{attribute addProperty BoxType "EK1960-2600-0021"}
{attribute addProperty Id "FSoE_CommandUSINT811FSOUT_Module_1_Module_FaultBIT10.1251FSOUT_Module_2_Module_FaultBIT10.1251FSOUT_Module_3_Module_FaultBIT10.1251FSOUT_Module_4_Module_FaultBIT10.1251FSOUT_Module_5_Module_FaultBIT10.1251FSOUT_Module_6_Module_FaultBIT10.1251FSOUT_Relais_Module_Module_FaultBIT10.1251FSIN_Module_1_Channel_1_Input_X6_1BIT10.1251FSIN_Module_1_Channel_2_Input_X6_2BIT10.1252FSIN_Module_1_Module_FaultBIT10.1251FSIN_Module_2_Channel_1_Input_X6_3BIT10.1251FSIN_Module_2_Channel_2_Input_X6_4BIT10.1252FSIN_Module_2_Module_FaultBIT10.1251FSIN_Module_3_Channel_1_Input_X6_5BIT10.1251FSIN_Module_3_Channel_2_Input_X6_6BIT10.1252FSIN_Module_3_Module_FaultBIT10.1251FSoE_CRC_000UINT1623FSIN_Module_4_Channel_1_Input_X6_7BIT10.1251FSIN_Module_4_Channel_2_Input_X6_8BIT10.1252FSIN_Module_4_Module_FaultBIT10.1251FSIN_Module_5_Channel_1_Input_X6_9BIT10.1251FSIN_Module_5_Channel_2_Input_X6_10BIT10.1252FSIN_Module_5_Module_FaultBIT10.1251FSIN_Module_6_Channel_1_Input_X8_1BIT10.1251FSIN_Module_6_Channel_2_Input_X8_2BIT10.1252FSIN_Module_6_Module_FaultBIT10.1251FSIN_Module_7_Channel_1_Input_X8_3BIT10.1251FSIN_Module_7_Channel_2_Input_X8_4BIT10.1252FSIN_Module_7_Module_FaultBIT10.1251FSIN_Module_8_Channel_1_Input_X8_5BIT10.1251FSIN_Module_8_Channel_2_Input_X8_6BIT10.1252FSIN_Module_8_Module_FaultBIT10.1251FSIN_Module_9_Channel_1_Input_X8_7BIT10.1251FSoE_CRC_001UINT1624FSIN_Module_9_Channel_2_Input_X8_8BIT10.1252FSIN_Module_9_Module_Fault_1BIT10.1251FSIN_Module_9_Module_Fault_2BIT10.1252FSIN_Module_10_Channel_1_Input_X8_9BIT10.1251FSIN_Module_10_Channel_2_Input_X8_10BIT10.1252FSIN_Module_10_Module_Fault_1BIT10.1251FSIN_Module_10_Module_Fault_2BIT10.1252FSoE_CRC_002UINT1625FSoE_Connection_IDUINT1622"}
{attribute addProperty CRC "994554049"}
{attribute addProperty SizeInBites "120"}
{attribute addProperty SizeInBytes "15"}
TYPE FSOE_3B47B0C1 :
STRUCT
	{attribute addProperty Name "FSoE_Command"}
	FSoE_Command : USINT;
	{attribute addProperty Name "FSOUT_Module_1_Module_Fault"}
	FSOUT_Module_1_Module_Fault : BOOL;
	{attribute addProperty Name "FSOUT_Module_2_Module_Fault"}
	FSOUT_Module_2_Module_Fault : BOOL;
	{attribute addProperty Name "FSOUT_Module_3_Module_Fault"}
	FSOUT_Module_3_Module_Fault : BOOL;
	{attribute addProperty Name "FSOUT_Module_4_Module_Fault"}
	FSOUT_Module_4_Module_Fault : BOOL;
	{attribute addProperty Name "FSOUT_Module_5_Module_Fault"}
	FSOUT_Module_5_Module_Fault : BOOL;
	{attribute addProperty Name "FSOUT_Module_6_Module_Fault"}
	FSOUT_Module_6_Module_Fault : BOOL;
	{attribute addProperty Name "FSOUT_Relais_Module_Module_Fault"}
	FSOUT_Relais_Module_Module_Fault : BOOL;
	{attribute addProperty Name "FSIN_Module_1_Channel_1_Input_X6_1"}
	FSIN_Module_1_Channel_1_Input_X6_1 : BOOL;
	{attribute addProperty Name "FSIN_Module_1_Channel_2_Input_X6_2"}
	FSIN_Module_1_Channel_2_Input_X6_2 : BOOL;
	{attribute addProperty Name "FSIN_Module_1_Module_Fault"}
	FSIN_Module_1_Module_Fault : BOOL;
	{attribute addProperty Name "FSIN_Module_2_Channel_1_Input_X6_3"}
	FSIN_Module_2_Channel_1_Input_X6_3 : BOOL;
	{attribute addProperty Name "FSIN_Module_2_Channel_2_Input_X6_4"}
	FSIN_Module_2_Channel_2_Input_X6_4 : BOOL;
	{attribute addProperty Name "FSIN_Module_2_Module_Fault"}
	FSIN_Module_2_Module_Fault : BOOL;
	{attribute addProperty Name "FSIN_Module_3_Channel_1_Input_X6_5"}
	FSIN_Module_3_Channel_1_Input_X6_5 : BOOL;
	{attribute addProperty Name "FSIN_Module_3_Channel_2_Input_X6_6"}
	FSIN_Module_3_Channel_2_Input_X6_6 : BOOL;
	{attribute addProperty Name "FSIN_Module_3_Module_Fault"}
	FSIN_Module_3_Module_Fault : BOOL;
	{attribute addProperty Name "FSoE_CRC_000"}
	FSoE_CRC_000 : UINT;
	{attribute addProperty Name "FSIN_Module_4_Channel_1_Input_X6_7"}
	FSIN_Module_4_Channel_1_Input_X6_7 : BOOL;
	{attribute addProperty Name "FSIN_Module_4_Channel_2_Input_X6_8"}
	FSIN_Module_4_Channel_2_Input_X6_8 : BOOL;
	{attribute addProperty Name "FSIN_Module_4_Module_Fault"}
	FSIN_Module_4_Module_Fault : BOOL;
	{attribute addProperty Name "FSIN_Module_5_Channel_1_Input_X6_9"}
	FSIN_Module_5_Channel_1_Input_X6_9 : BOOL;
	{attribute addProperty Name "FSIN_Module_5_Channel_2_Input_X6_10"}
	FSIN_Module_5_Channel_2_Input_X6_10 : BOOL;
	{attribute addProperty Name "FSIN_Module_5_Module_Fault"}
	FSIN_Module_5_Module_Fault : BOOL;
	{attribute addProperty Name "FSIN_Module_6_Channel_1_Input_X8_1"}
	FSIN_Module_6_Channel_1_Input_X8_1 : BOOL;
	{attribute addProperty Name "FSIN_Module_6_Channel_2_Input_X8_2"}
	FSIN_Module_6_Channel_2_Input_X8_2 : BOOL;
	{attribute addProperty Name "FSIN_Module_6_Module_Fault"}
	FSIN_Module_6_Module_Fault : BOOL;
	{attribute addProperty Name "FSIN_Module_7_Channel_1_Input_X8_3"}
	FSIN_Module_7_Channel_1_Input_X8_3 : BOOL;
	{attribute addProperty Name "FSIN_Module_7_Channel_2_Input_X8_4"}
	FSIN_Module_7_Channel_2_Input_X8_4 : BOOL;
	{attribute addProperty Name "FSIN_Module_7_Module_Fault"}
	FSIN_Module_7_Module_Fault : BOOL;
	{attribute addProperty Name "FSIN_Module_8_Channel_1_Input_X8_5"}
	FSIN_Module_8_Channel_1_Input_X8_5 : BOOL;
	{attribute addProperty Name "FSIN_Module_8_Channel_2_Input_X8_6"}
	FSIN_Module_8_Channel_2_Input_X8_6 : BOOL;
	{attribute addProperty Name "FSIN_Module_8_Module_Fault"}
	FSIN_Module_8_Module_Fault : BOOL;
	{attribute addProperty Name "FSIN_Module_9_Channel_1_Input_X8_7"}
	FSIN_Module_9_Channel_1_Input_X8_7 : BOOL;
	{attribute addProperty Name "FSoE_CRC_001"}
	FSoE_CRC_001 : UINT;
	{attribute addProperty Name "FSIN_Module_9_Channel_2_Input_X8_8"}
	FSIN_Module_9_Channel_2_Input_X8_8 : BOOL;
	{attribute addProperty Name "FSIN_Module_9_Module_Fault_1"}
	FSIN_Module_9_Module_Fault_1 : BOOL;
	{attribute addProperty Name "FSIN_Module_9_Module_Fault_2"}
	FSIN_Module_9_Module_Fault_2 : BOOL;
	{attribute addProperty Name "FSIN_Module_10_Channel_1_Input_X8_9"}
	FSIN_Module_10_Channel_1_Input_X8_9 : BOOL;
	{attribute addProperty Name "FSIN_Module_10_Channel_2_Input_X8_10"}
	FSIN_Module_10_Channel_2_Input_X8_10 : BOOL;
	{attribute addProperty Name "FSIN_Module_10_Module_Fault_1"}
	FSIN_Module_10_Module_Fault_1 : BOOL;
	{attribute addProperty Name "FSIN_Module_10_Module_Fault_2"}
	FSIN_Module_10_Module_Fault_2 : BOOL;
	{attribute 'hide'}
	reserve_1_BIT_0 : BOOL;
	{attribute 'hide'}
	reserve_1_BIT_1 : BOOL;
	{attribute 'hide'}
	reserve_1_BIT_2 : BOOL;
	{attribute 'hide'}
	reserve_1_BIT_3 : BOOL;
	{attribute 'hide'}
	reserve_1_BIT_4 : BOOL;
	{attribute 'hide'}
	reserve_1_BIT_5 : BOOL;
	{attribute 'hide'}
	reserve_1_BIT_6 : BOOL;
	{attribute 'hide'}
	reserve_1_BIT_7 : BOOL;
	{attribute 'hide'}
	reserve_1_BIT_8 : BOOL;
	{attribute addProperty Name "FSoE_CRC_002"}
	FSoE_CRC_002 : UINT;
	{attribute addProperty Name "FSoE_Connection_ID"}
	FSoE_Connection_ID : UINT;
END_STRUCT
END_TYPE

(* stored: Version 1.2.0.0, ProductVersion 3.1.4024.9
   DUT FSOE_3B47B0C1: Id {5de64ecb-5170-4f93-a7dd-85782f79679f} *)
